FUNCTION_BLOCK FB_SQLExpert_InsertBuffer
// Fonctionnement : Tableau de 2000 structures en input. Dès qu'on atteint 1000 structures remplies, décalage de l'espace mémoire
// pour en 1 temps de cycle pour ne pas perdre de données sur le transfert.
VAR CONSTANT
	CstNbLigneBuffer		: DINT:= 250;
	CstNbLigneBufferMax	 	: DINT:= 5000;

END_VAR

VAR_INPUT
	NomTable				: STRING := 'Table100ms';
	hDBID					: UDINT;
END_VAR

VAR_OUTPUT
	OUT_Error				: BOOL;
	OUT_Busy				: BOOL;
END_VAR

VAR
	ETAPE					: UINT;

    myStruct      			: ARRAY[1..CstNbLigneBuffer] OF St_DataHisto;
	myStructMax    			: ARRAY[1..CstNbLigneBufferMax] OF St_DataHisto;
	StructNull				: St_DataHisto;

    SQLDatabase				: FB_SQLDatabaseEvt('',T#10S);
	SQLCommand1				: FB_SQLCommandEvt('',T#10S);
	SQLCommandNull			: FB_SQLCommandEvt('',T#10S);
	bConnected				: BOOL;              	        	

	TrameValues				: T_MaxString := ' ([Timestamp],[Timestamp_Ms],[ParentId],[Value])';
	pPosRequete				: DINT;                		
	RequeteFinale			: ARRAY[1..100] OF STRING(1000);	
	RequeteFinaleNull		: ARRAY[1..100] OF STRING(1000);	
	sTimeStamp				: STRING(255);               	
	RequeteEntete			: STRING(1000);
	sInsertValue			: STRING(1000);
	Format					: FB_FormatString;
	                		
	NbElemBuffer			: DINT;
	KK						: DINT;
	                    	
	CmdStart				: BOOL;
	TrigCmdExec				: R_TRIG;
	TrigStart				: R_TRIG;
	RsStart					: RS;
	
	// Insert
		hDBID_BaseTampon	: UINT := 3;
	// AlarmManagement      
		bBufferMaxFull 		: BOOL;        		
		bInStructNull		: BOOL;
		
		
		
	
END_VAR

NbElemBuffer := M_Count();
CmdStart := NbElemBuffer>= CstNbLigneBuffer;


TrigStart(CLK := CmdStart);
IF TrigStart.Q THEN
	FOR KK := 1 TO CstNbLigneBuffer DO
		myStruct[KK] := myStructMax[KK];
	END_FOR
END_IF


// call functionblock

CASE ETAPE OF
	0://INITIALISATION  & CONNECTION
		RequeteEntete := concat(concat('INSERT INTO ',NomTable),concat(TrameValues,' VALUES '));
		RsStart(SET := TrigStart.Q);
		IF RsStart.Q1 THEN
			IF SQLDatabase.Connect(hDBID := hDBID) THEN;
				bConnected := NOT sqldatabase.bError;
				IF bConnected THEN
					ETAPE := 1;
				ELSE
					ETAPE := 255;
				END_IF
			END_IF
		END_IF
		
	1: // CONNECTED
		IF SQLDatabase.CreateCmd(pSQLCommand := ADR(SQLCommand1)) THEN 
			IF NOT SQLCommand1.bError THEN
				ETAPE := 2;
			ELSIF SQLCommand1.bError THEN
				ETAPE := 255;
			END_IF
		END_IF
	2:
		MEMCPY(srcAddr:= ADR(RequeteEntete), destAddr := ADR(requeteFinale), n:= SIZEOF(RequeteEntete));
		pPosRequete := LEN(STR := RequeteEntete);
		FOR KK:= 1 TO CstNbLigneBuffer-1 DO
			sTimeStamp	:= right(STR := DT_TO_STRING(myStruct[KK].Timestamp), SIZE := LEN(DT_TO_STRING(myStruct[KK].Timestamp))-3);
			Format(sFormat := '($'%s $',%.3d,%.4d,%5.2f),', arg1 := F_STRING(sTimeStamp),arg2:=F_DINT(myStruct[KK].Timestamp_Ms), arg3:= F_DINT(myStruct[KK].ParentId), arg4:= F_LREAL(myStruct[KK].Value), sOut=>sInsertValue);
			MEMCPY(srcAddr:= ADR(sInsertValue), destAddr := ADR(requeteFinale)+DINT_TO_DWORD(pPosRequete), n:= SIZEOF(sInsertValue));
			pPosRequete:= pPosRequete + LEN(STR := sInsertValue);
		END_FOR
		sTimeStamp	:= right(STR := DT_TO_STRING(myStruct[KK].Timestamp), SIZE := LEN(DT_TO_STRING(myStruct[KK].Timestamp))-3);
		Format(sFormat := '($'%s $',%.3d,%.4d,%5.2f)', arg1 := F_STRING(sTimeStamp),arg2:=F_DINT(myStruct[KK].Timestamp_Ms), arg3:= F_DINT(myStruct[KK].ParentId), arg4:= F_LREAL(myStruct[KK].Value), sOut=>sInsertValue);
		MEMCPY(srcAddr:= ADR(sInsertValue), destAddr := ADR(requeteFinale)+DINT_TO_DWORD(pPosRequete), n:= SIZEOF(sInsertValue));
	
		IF SQLCommand1.Execute(pSQLCmd := ADR(RequeteFinale), cbSQLCmd := SIZEOF(Requetefinale))THEN
			
			IF  NOT SQLCommand1.bError THEN
				ETAPE := 3;
			ELSIF SQLCommand1.bError THEN
				ETAPE := 255;
			END_IF
		END_IF
	3:
			IF SQLDatabase.Disconnect() THEN
				ETAPE := 4;
			END_IF 
	4:
		IF NOT SQLDatabase.bError THEN
			RequeteFinale := RequeteFinaleNull;
			FOR KK := CstNbLigneBuffer TO CstNbLigneBufferMax -1 DO
				myStructMax[KK+1-CstNbLigneBuffer]:= myStructMax[KK+1];
			END_FOR
			
			FOR KK := CstNbLigneBufferMax-CstNbLigneBuffer+1 TO CstNbLigneBufferMax DO
				myStructMax[KK]:= StructNull;
			END_FOR			
			
			TrigStart(CLK := FALSE);
			RsStart(RESET1 := TRUE);
			RsStart(RESET1 := FALSE);
			TrigCmdExec(CLK := FALSE);
			CmdStart := FALSE;
			Etape := 0;
			OUT_Error := FALSE;
		ELSE 
			ETAPE := 255;
		END_IF
	255: 
		RequeteFinale := RequeteFinaleNull;
		OUT_Error := TRUE;
		Etape := 0;
		RsStart(RESET1 := TRUE);
		RsStart(RESET1 := FALSE);
		TrigCmdExec(CLK := FALSE);
		CmdStart := FALSE;
		
END_CASE

METHOD M_AddLine : BOOL
VAR_INPUT
	InStruct			: St_DataHisto;
END_VAR

VAR
END_VAR
// Check the biggest buffer isn't full
IF MEMCMP(pBuf1 := ADR(StructNull), pBuf2 := ADR(myStructMax[CstNbLigneBufferMax]), n := SIZEOF(StructNull)) <> 0 THEN
	bBufferMaxFull := TRUE;
ELSE
	//Check the input struct isn't null
	IF MEMCMP(pBuf1 := ADR(StructNull), pBuf2 := ADR(InStruct), n := SIZEOF(StructNull)) = 0 THEN
		bInStructNull := TRUE;
	ELSE
		// We parse the biggest buffer
		FOR KK := 1 TO CstNbLigneBufferMax DO 
			IF MEMCMP(pBuf1 := ADR(StructNull), pBuf2 := ADR(myStructMax[KK]), n := SIZEOF(StructNull)) = 0 THEN
				myStructMax[KK] := InStruct;
				bBufferMaxFull := FALSE;
				EXIT;
			END_IF
		END_FOR
	END_IF
END_IF
END_METHOD

METHOD M_AlarmManager : BOOL
VAR_INPUT
	AlarmCode : WORD;
	
END_VAR


AlarmCode.0 := bBufferMaxFull;
AlarmCode.1 := bInStructNull;
END_METHOD

METHOD M_Count : DINT
VAR_INPUT
END_VAR
VAR

END_VAR
FOR KK := 1 TO CstNbLigneBufferMax DO 

	IF MEMCMP(pBuf1 := ADR(StructNull), pBuf2 := ADR(myStructMax[KK]), n := SIZEOF(StructNull)) = 0 THEN
		EXIT ;
	END_IF
END_FOR

M_Count := MIN(KK, CstNbLigneBufferMax);
END_METHOD

END_FUNCTION_BLOCK

(* stored: Version 1.1.0.1, ProductVersion 3.1.4024.6
   POU FB_SQLExpert_InsertBuffer: Id {ab3c8a2a-18cd-4cdc-a3f7-169d78c10d35}, SpecialFunc None
   Method M_AddLine: Id {54ef9f07-82b0-4fb2-a64d-fba1cee4a9b1}
   Method M_AlarmManager: Id {830864cd-9ba0-4e70-a799-8914b3722edf}
   Method M_Count: Id {00f25f58-957d-4156-9716-1bbdf07e1518} *)
